FUNCTION_BLOCK UA_MethodCall_ADSWriteControlReq
VAR_INPUT
	bExecute			: BOOL;
	nConnectionHdl		: DWORD;
	nNamespaceIndex		: UINT; 		(* to be retrieved using UA_GetNamespaceIndex *)
	sNetID				: T_AmsNetId; 	(* AmsNetId OF the Target *)
	nPort				: INT; 			(* Port number	*)
	nAdsState			: DINT;			(* IndexGroup*)
	nDeviceState		: DINT; 		(* IndexOffset*)
	pWriteData			: PVOID;
	cbWriteData			: UDINT;		(* Count of bytes to be written*)
	Timeout				: TIME := DEFAULT_ADS_TIMEOUT;
END_VAR
VAR_OUTPUT
	bDone				: BOOL;
	bBusy				: BOOL;
	bError				: BOOL;
	nErrorID			: DWORD;
END_VAR
VAR
	iWriteControlReqState	: INT;
	RTrig					: R_TRIG;

	fbUA_MethodGetHandle: UA_MethodGetHandle;
	nMethodHdl			: DWORD;
	ObjectNodeID		: ST_UANodeID;
	MethodNodeID		: ST_UANodeID;

	fbUA_MethodCall		: UA_MethodCall;
	InputArguments		: ARRAY [1..nNumberOfInputArguments] OF ST_UAMethodArgInfo; (*WriteControlReq has 5 input parameters *)
	nNumberOfOutputArguments_R	: UDINT;
	nArg				: INT;
	nInputData			: ARRAY [1..nInputArgSize] OF BYTE;(* NetID(24)+ Port(2)+ ADSState(4)+ DeviceState(4)*)
	nOffset				: UDINT;
	
	fbUA_MethodReleaseHandle: UA_MethodReleaseHandle;
	bInputDataError 		: BOOL; 
END_VAR
VAR CONSTANT
	nInputArgSize			: UDINT := 34; // (* NetID(24)+ Port(2)+ ADSState(4)+ DeviceState(4)*)
	nNumberOfInputArguments : UDINT := 5;
	nNumberOfOutputArguments: UDINT := 0;
END_VAR

(*
ADSWriteControlReq(
******** Input Arguments ********
	string sNetID, 		: AmsNetId of the Target
	int16 Port,			: Port number	
	int32 AdsState,		: Ads State
	int32 DeviceState	: Device State
	ByteString Data		: Data to be written to the device
******** Output Arguments ********
	
);
*)
RTrig(CLK:= bExecute);

CASE iWriteControlReqState OF

0:	(* Get Method Handle *)
	IF RTrig.Q THEN
		bBusy		:= TRUE;
		bDone 		:= FALSE;
		bError		:= FALSE;
		nErrorID	:= 0;
		ObjectNodeID.eIdentifierType 	:= eUAIdentifierType_String;
		ObjectNodeID.nNamespaceIndex 	:= nNamespaceIndex;
		ObjectNodeID.sIdentifier		:= 'ADSAMS';
	
		MethodNodeID.eIdentifierType 	:= eUAIdentifierType_String;
		MethodNodeID.nNamespaceIndex 	:= nNamespaceIndex;
		MethodNodeID.sIdentifier		:= 'ADSAMS.AdsWriteControlReq';

		M_Init();
		IF bInputDataError = FALSE THEN
			iWriteControlReqState 	:= iWriteControlReqState + 1;
		ELSE
			bBusy		:= FALSE;
			bError 		:= TRUE;
			nErrorID 	:= DEVICE_INVALIDSIZE; //16#705 parameter size not correct
		END_IF		
	END_IF


1:	(* Method Get Handle *)
	fbUA_MethodGetHandle(
			Execute			:= TRUE,
			ConnectionHdl	:= nConnectionHdl,
			ObjectNodeID	:= ObjectNodeID,
			MethodNodeID 	:= MethodNodeID,
			Timeout			:= Timeout,
			MethodHdl		=> nMethodHdl
		);
	IF NOT fbUA_MethodGetHandle.Busy THEN
		fbUA_MethodGetHandle(Execute := FALSE);

		IF NOT fbUA_MethodGetHandle.Error THEN
			(*  *)
			iWriteControlReqState := iWriteControlReqState + 1; (* Call Method *)
		ELSE
			bError			:= TRUE;
			nErrorID		:= fbUA_MethodGetHandle.ErrorID;
			iWriteControlReqState 	:= 3; (* Release Handle *)
		END_IF
	END_IF


2:	(* Method Call *)
	fbUA_MethodCall(
		Execute					:= TRUE,
		ConnectionHdl			:= nConnectionHdl,
		MethodHdl				:= nMethodHdl,
		nNumberOfInputArguments := nNumberOfInputArguments,		(* 5 *)
		pInputArgInfo			:= ADR(InputArguments),
		cbInputArgInfo			:= SIZEOF(InputArguments),
		pInputArgData			:= ADR(nInputData),
		cbInputArgData			:= nOffset,
		pInputWriteData			:= pWriteData,
		cbInputWriteData		:= cbWriteData,
		nNumberOfOutputArguments:= nNumberOfOutputArguments,		(* 0 *)
		pOutputArgInfo			:= 0,
		cbOutputArgInfo			:= 0,
		pOutputArgInfoAndData	:= ADR(nNumberOfOutputArguments_R),	//minimum output
		cbOutputArgInfoAndData	:= SIZEOF(nNumberOfOutputArguments_R),	//minimum output
		Timeout					:= Timeout
	);

	IF NOT fbUA_MethodCall.Busy THEN
		fbUA_MethodCall(Execute := FALSE);
		IF NOT fbUA_MethodCall.Error THEN
			(*  *)
			iWriteControlReqState 	:= iWriteControlReqState + 1; (* Release handle *)
			(*MEMSET(ADR(Data),0,nMaxNumberofOutputArgBytes);
			MEMCPY(ADR(Data),ADR(OutputArguments),cbData); *)
		ELSE
			bError					:= TRUE;
			nErrorID				:= fbUA_MethodCall.ErrorID;
			iWriteControlReqState	:= 3; (* Release handle *)
		END_IF
	END_IF


3:	(* Release Method Handle *)
	fbUA_MethodReleaseHandle(
		Execute			:= TRUE,
		ConnectionHdl	:= nConnectionHdl,
		MethodHdl		:= nMethodHdl,
		Timeout			:= Timeout
	);

	IF NOT fbUA_MethodReleaseHandle.Busy THEN
		fbUA_MethodReleaseHandle(Execute := FALSE);
		bBusy := FALSE;
		IF NOT fbUA_MethodReleaseHandle.Error THEN
			(* session closed *)
			bDone := TRUE;
			iWriteControlReqState 	:= 0; (* idle *)
		ELSE
			bError			:= TRUE;
			nErrorID		:= fbUA_MethodReleaseHandle.ErrorID;
			iWriteControlReqState 	:= 0; (* idle *)
		END_IF
	END_IF
END_CASE

ACTION M_Init:
bInputDataError := FALSE; 
nOffset := 0;
MEMSET(ADR(InputArguments),0,SIZEOF(InputArguments));
MEMSET(ADR(nInputData),0,SIZEOF(nInputData));

nArg := 1;
(*sNetID := sAmsNetID;*)	(********** NET ID **********);
InputArguments[nArg].DataType			:= eUAType_String;
InputArguments[nArg].ValueRank			:= -1; 							(* Scalar = -1 or Array *)
InputArguments[nArg].ArrayDimensions[1]	:= 0; 							(* Number of Dimension in case its an array *)
InputArguments[nArg].nLenData			:= INT_TO_UDINT(LEN(sNetId)) + 1;				(* Length if its a STRING *)
IF nOffset + INT_TO_UDINT(LEN(sNetId))+1 > nInputArgSize THEN 
	bInputDataError := TRUE;
	RETURN;
ELSE
	MEMCPY(ADR(nInputData)+nOffset,ADR(sNetId),INT_TO_UDINT(LEN(sNetId))+1);				(* VALUE in BYTES FORM *)
	nOffset := nOffset + INT_TO_UDINT(LEN(sNetId))+1;
END_IF

nArg := nArg + 1;
(* nPort := 851;*)			(********** PORT **********)
InputArguments[nArg].DataType			:= eUAType_Int16;
InputArguments[nArg].ValueRank			:= -1; 							(* Scalar = -1 or Array *)
InputArguments[nArg].ArrayDimensions[1]	:= 0; 							(* Number of Dimension in case its an array *)
InputArguments[nArg].nLenData			:= SIZEOF(nPort);				(* Length if its a STRING *)
IF nOffset + SIZEOF(nPort) > nInputArgSize THEN 
	bInputDataError := TRUE;
	RETURN;
ELSE
	MEMCPY(ADR(nInputData)+nOffset,ADR(nPort),SIZEOF(nPort));			(* VALUE in BYTES FORM *)
	nOffset := nOffset + SIZEOF(nPort);
END_IF

nArg := nArg + 1;
(*nAdsState := ;*)	(********** Ads State **********)
InputArguments[nArg].DataType			:= eUAType_Int32;
InputArguments[nArg].ValueRank			:= -1; 							(* Scalar = -1 or Array *)
InputArguments[nArg].ArrayDimensions[1]	:= 0; 							(* Number of Dimension in case its an array *)
InputArguments[nArg].nLenData			:= SIZEOF(nAdsState);			(* Length if its a STRING *)
IF nOffset + SIZEOF(nAdsState) > nInputArgSize THEN 
	bInputDataError := TRUE;
	RETURN;
ELSE
	MEMCPY(ADR(nInputData)+nOffset,ADR(nAdsState),SIZEOF(nAdsState));		(* VALUE in BYTES FORM *)
	nOffset := nOffset + SIZEOF(nAdsState);
END_IF

nArg := nArg + 1;
(*nDeviceState := ; *)		(********** Device State **********)
InputArguments[nArg].DataType			:= eUAType_Int32;
InputArguments[nArg].ValueRank			:= -1; 							(* Scalar = -1 or Array *)
InputArguments[nArg].ArrayDimensions[1]	:= 0; 							(* Number of Dimension in case its an array *)
InputArguments[nArg].nLenData			:= SIZEOF(nDeviceState);		(* Length if its a STRING *)
IF nOffset + SIZEOF(nDeviceState) > nInputArgSize THEN 
	bInputDataError := TRUE;
	RETURN;
ELSE
	MEMCPY(ADR(nInputData)+nOffset,ADR(nDeviceState),SIZEOF(nDeviceState));	(* VALUE in BYTES FORM *)
	nOffset := nOffset + SIZEOF(nDeviceState);
END_IF

nArg := nArg + 1;
(*Data := ; *)		(*********** WriteData ***********)
InputArguments[nArg].DataType			:= eUAType_ByteString;
InputArguments[nArg].ValueRank			:= -1; 							(* Scalar = -1 or Array *)
InputArguments[nArg].ArrayDimensions[1]	:= 0; 							(* Number of Dimension in case its an array *)
InputArguments[nArg].nLenData			:= cbWriteData;						(* Length if its a STRING *)
END_ACTION

END_FUNCTION_BLOCK

(* stored: Version 1.1.0.1, ProductVersion 3.1.4022.6
   POU UA_MethodCall_ADSWriteControlReq: Id {862eb0ba-9983-47a1-8542-b74349889a8d}, SpecialFunc None
   Action M_Init: Id {e0797451-b58e-4d91-8325-addef3b0f1bf} *)
